TYPE ST_HE_SolidAttenuatorSlotSettings :
STRUCT
    bEnabled : BOOL;
END_STRUCT
END_TYPE

(* stored: Version 1.1.0.1
   DUT ST_HE_SolidAttenuatorSlotSettings: Id {34a02836-e654-4aa3-bf7f-f34baf13f071} *)
